// TIA Portal V19 export
TYPE "LAF_typePlasticWorkstationEm5Parameters"
// stored: Access Published
   STRUCT
      cm1Vfd208 : "LAF_typeVfdParameters";
      cm4SR1000 { S7_SetPoint := 'True'} : "LAF_typeSR1000Parameters";
   END_STRUCT;
END_TYPE
